Fanuc KAREL source: kb00163.KL

-- PROVISIONAL review KL for V1013-1; original PC SHA256 e8f2613238712ed0d6846f8f8402f98f011ccc7eae795fbeb94284d556b23ca8
-- Incomplete behavior may be omitted. Consult companion uncertainty JSON. Do not deploy.
PROGRAM KB00163
%NOLOCKGROUP
BEGIN
  -- UNRESOLVED_PC offsets 5-12; opcodes 9D,23
  -- UNRESOLVED_PC offsets 17-35; opcodes 27,22,22,27,9D,31
  -- UNRESOLVED_PC offsets 40-44; opcodes 7F
END KB00163
